FUNCTION_BLOCK FB_DisplacementControl_SC 
VAR_INPUT
	
	fDisplacementNormalizedInput 	: LREAL;
	bEnable 						: BOOL; 
	fYokeNormalizedFeedback 		: LREAL;
	
	fVelRef							: LREAL;
	
END_VAR
VAR_OUTPUT
	fNormalizedOutput 				: LREAL; 
END_VAR

VAR PERSISTENT
	
END_VAR

VAR
	fProportionalGain 				: LREAL;
	fIntegralGain					: LREAL;
	fDerivateGain					: LREAL;	


	fbPID_SC						: FB_PID_SC;
	fbPID_new						: FB_PID_Controller;
	fYoke_error						: LREAL;
	fProportinalGain_output			: LREAL;
	fIntegralGain_output			: LREAL;
	fDerivateGain_output			: LREAL;
END_VAR

IF bEnable THEN
	


IF fVelRef > 0.0 THEN
	fProportionalGain := G_Engineer_HMI.fPGain_IL_Pos;
	fIntegralGain := G_Engineer_HMI.fIGain_IL_Pos;
	fDerivateGain := G_Engineer_HMI.fDGain_IL_Pos;
ELSIF fVelRef < 0.0 THEN
	fProportionalGain := G_Engineer_HMI.fPGain_IL_Neg;
	fIntegralGain := G_Engineer_HMI.fIGain_IL_Neg;
	fDerivateGain := G_Engineer_HMI.fDGain_IL_Neg;
ELSE
	fProportionalGain := G_Engineer_HMI.fPGain_IL_Pos;
	fIntegralGain := G_Engineer_HMI.fIGain_IL_Pos;
	fDerivateGain := G_Engineer_HMI.fDGain_IL_Pos;
END_IF

		
		fbPID_SC(
	ssMethodType := BOOL_TO_SINT(bEnable),
	fSignalReference := fDisplacementNormalizedInput,
	fSignalFeedback := fYokeNormalizedFeedback,
	fProportionalGain := fProportionalGain,
	fIntegralGain := fIntegralGain,
	bActivateIntegralControl := G_Engineer_HMI.bIenable_IL,
	bEnable := bEnable,
	bIntegralControlReset := FALSE,
	bActivateDerivativeControl := FALSE,
	fDerivativeGain := fDerivateGain,
	fClosedLoopSignal => fNormalizedOutput,
	fSignalError =>G_PID_Tuning.fYoke_error,
	P_out => G_PID_Tuning.fProportinalGain_output_dis,
	I_out => G_PID_Tuning.fIntegralGain_output_dis,
	D_out => G_PID_Tuning.fDerivateGain_output_dis
	);	


	//Make Output global for plot
	G_PID_Tuning.PID_output_dis := fNormalizedOutput;
	
ELSE 
	fNormalizedOutput := 0.0; // Ingen output uten aktivering
END_IF

END_FUNCTION_BLOCK

(* stored: Version 1.1.0.1
   POU FB_DisplacementControl_SC: Id {bdc1fc63-8ad7-4439-bfe4-2ff7f2a8ff55}, SpecialFunc None *)
